Omron Sysmac Studio project comodo-sync-lib (Sysmac Studio 1.64.0.64008, LibraryProject)

# Controller new_Controller_0: NX102-9020 version 1.50
Task PrimaryTask (priority 4, period or condition 2000): Program0

VAR_GLOBAL
    Robot_Positions : ARRAY[0..5] OF LREAL;
    Robot_In : LWORD;  (* network input *)
    Robot_Out : LWORD;  (* network output *)
    In_Joint_1 : LREAL;  (* published *)
    In_Joint_2 : LREAL;  (* published *)
    In_Joint_3 : LREAL;  (* published *)
    In_Joint_4 : LREAL;  (* published *)
    In_Joint_5 : LREAL;  (* published *)
    In_Joint_6 : LREAL;  (* published *)
    Out_Joint_1 : LREAL;  (* published *)
    Out_Joint_2 : LREAL;  (* published *)
    Out_Joint_3 : LREAL;  (* published *)
    Out_Joint_4 : LREAL;  (* published *)
    Out_Joint_5 : LREAL;  (* published *)
    Out_Joint_6 : LREAL;  (* published *)
    Is_Monitoring : BOOL;
    Is_Moving_Linear : BOOL;
END_VAR

PROGRAM Program0
VAR
    test : BOOL;
END_VAR

(* Section Section0: ladder, written here as Structured Text *)

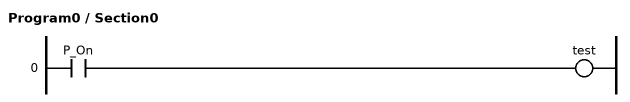
(* Rung 0 *)
test := P_On;
END_PROGRAM

FUNCTION MapLREAL : LREAL
VAR_INPUT
    Num : LREAL;
    In_Min : LREAL;
    In_Max : LREAL;
    Out_Min : LREAL;
    Out_Max : LREAL;
END_VAR
MapLREAL := (Num - In_Min) * (Out_Max - Out_Min) / (In_Max - In_Min) + Out_Min;
END_FUNCTION

FUNCTION ReceiveRobotPositions : BOOL
VAR_EXTERNAL
    Robot_Positions : ARRAY[0..5] OF LREAL;
    In_Joint_1 : LREAL;
    In_Joint_2 : LREAL;
    In_Joint_3 : LREAL;
    In_Joint_4 : LREAL;
    In_Joint_5 : LREAL;
    In_Joint_6 : LREAL;
END_VAR
IF In_Joint_1 <> Robot_Positions[0] THEN
	In_Joint_1 := Robot_Positions[0];
END_IF;
IF In_Joint_2 <> Robot_Positions[1] THEN
	In_Joint_2 := Robot_Positions[1];
END_IF;
IF In_Joint_3 <> Robot_Positions[2] THEN
	In_Joint_3 := Robot_Positions[2];
END_IF;
IF In_Joint_4 <> Robot_Positions[3] THEN
	In_Joint_4 := Robot_Positions[3];
END_IF;
IF In_Joint_5 <> Robot_Positions[4] THEN
	In_Joint_5 := Robot_Positions[4];
END_IF;
IF In_Joint_6 <> Robot_Positions[5] THEN
	In_Joint_6 := Robot_Positions[5];
END_IF;
END_FUNCTION

FUNCTION SendPositionsToRobot : BOOL
VAR
    Temp_Output : LWORD;
    Temp_Bits : LWORD;
    Shifted_Bits : LWORD;
END_VAR
VAR CONSTANT
    Movement_Bit : LWORD := 16#2000000000000000;
    Monitor_Bit : LWORD := 16#1000000000000000;
END_VAR
VAR_EXTERNAL
    Robot_Positions : ARRAY[0..5] OF LREAL;
    Robot_In : LWORD;
    Out_Joint_1 : LREAL;
    Out_Joint_2 : LREAL;
    Out_Joint_3 : LREAL;
    Out_Joint_4 : LREAL;
    Out_Joint_5 : LREAL;
    Out_Joint_6 : LREAL;
    Is_Moving_Linear : BOOL;
    Is_Monitoring : BOOL;
END_VAR
Robot_Positions[0] := Out_Joint_1;
Robot_Positions[1] := Out_Joint_2;
Robot_Positions[2] := Out_Joint_3;
Robot_Positions[3] := Out_Joint_4;
Robot_Positions[4] := Out_Joint_5;
Robot_Positions[5] := Out_Joint_6;

Temp_Output := 16#0;

Temp_Bits := LREAL_TO_LWORD(MapLREAL(Robot_Positions[0], -230.0, 230.0, 0.0, 1023.0));
Temp_Output := Temp_Output OR Temp_Bits;


Temp_Bits := LREAL_TO_LWORD(MapLREAL(Robot_Positions[1], -115.0, 113.0, 0.0, 1023.0));
Shifted_Bits := SHL(Temp_Bits, 10);
Temp_Output := Temp_Output OR Shifted_Bits;


Temp_Bits := LREAL_TO_LWORD(MapLREAL(Robot_Positions[2], -205.0, 55.0, 0.0, 1023.0));
Shifted_Bits := SHL(Temp_Bits, 20);
Temp_Output := Temp_Output OR Shifted_Bits;


Temp_Bits := LREAL_TO_LWORD(MapLREAL(Robot_Positions[3], -230.0, 230.0, 0.0, 1023.0));
Shifted_Bits := SHL(Temp_Bits, 30);
Temp_Output := Temp_Output OR Shifted_Bits;


Temp_Bits := LREAL_TO_LWORD(MapLREAL(Robot_Positions[4], -125.0, 120.0, 0.0, 1023.0));
Shifted_Bits := SHL(Temp_Bits, 40);
Temp_Output := Temp_Output OR Shifted_Bits;


Temp_Bits := LREAL_TO_LWORD(MapLREAL(Robot_Positions[5], -400.0, 400.0, 0.0, 1023.0));
Shifted_Bits := SHL(Temp_Bits, 50);
Temp_Output := Temp_Output OR Shifted_Bits;

IF Is_Monitoring THEN 
		Temp_Output := Temp_Output OR Monitor_Bit;
ELSE
		Temp_Output := Temp_Output AND (NOT Monitor_Bit);
END_IF;

IF Is_Moving_Linear THEN
		Temp_Output := Temp_Output OR Movement_Bit;
ELSE
		Temp_Output := Temp_Output AND (NOT Movement_Bit);
END_IF;

Robot_In := Temp_Output;
END_FUNCTION

FUNCTION ChangeState : BOOL
VAR
    Previous_Monitor_State : BOOL;
    Temp_Output : LWORD;
END_VAR
VAR CONSTANT
    Monitor_Bit : LWORD := 16#1000000000000000;
END_VAR
VAR
    Previous_Movement_State : BOOL;
END_VAR
VAR CONSTANT
    Movement_Bit : LWORD := 16#2000000000000000;
END_VAR
VAR_EXTERNAL
    Is_Monitoring : BOOL;
    Robot_Out : LWORD;
    Robot_In : LWORD;
    Is_Moving_Linear : BOOL;
END_VAR
IF Is_Monitoring <> Previous_Monitor_State OR Is_Moving_Linear <> Previous_Movement_State THEN
	Temp_Output := Robot_In;
	IF Is_Monitoring THEN 
		Temp_Output := Temp_Output OR Monitor_Bit;
	ELSE
		Temp_Output := Temp_Output AND (NOT Monitor_Bit);
	END_IF;
	
	IF Is_Moving_Linear THEN
		Temp_Output := Temp_Output OR Movement_Bit;
	ELSE
		Temp_Output := Temp_Output AND (NOT Movement_Bit);
	END_IF;
		
	Previous_Monitor_State := Is_Monitoring;
	Previous_Movement_State := Is_Moving_Linear;
	
	Robot_In := Temp_Output;
END_IF;
END_FUNCTION

FUNCTION_BLOCK ParseRobotData
VAR
    value : UINT;
    shifted_input : LWORD;
END_VAR
VAR_INPUT
    IN : BOOL;
END_VAR
VAR_EXTERNAL
    Robot_Positions : ARRAY[0..5] OF LREAL;
    Robot_Out : LWORD;
END_VAR
value := LWORD_TO_UINT(Robot_Out AND LWORD#16#3FF);
Robot_Positions[0] :=MapLREAL(value, 0.0, 1023.0, -230.0, 230.0);

shifted_input := SHR(Robot_Out, 10);
value := LWORD_TO_UINT(shifted_input AND LWORD#16#3FF);
Robot_Positions[1]:=MapLREAL(value, 0.0, 1023.0, -115.0, 113.0);

shifted_input := SHR(Robot_Out, 20);
value := LWORD_TO_UINT(shifted_input AND LWORD#16#3FF);
Robot_Positions[2]:=MapLREAL(value, 0.0, 1023.0, -205.0, 55.0);

shifted_input := SHR(Robot_Out, 30);
value := LWORD_TO_UINT(shifted_input AND LWORD#16#3FF);
Robot_Positions[3]:=MapLREAL(value, 0.0, 1023.0, -230.0, 230.0);

shifted_input := SHR(Robot_Out, 40);
value := LWORD_TO_UINT(shifted_input AND LWORD#16#3FF);
Robot_Positions[4]:=MapLREAL(value, 0.0, 1023.0, -125.0, 120.0);

shifted_input := SHR(Robot_Out, 50);
value := LWORD_TO_UINT(shifted_input AND LWORD#16#3FF);
Robot_Positions[5]:=MapLREAL(value, 0.0, 1023.0, -400.0, 400.0);
END_FUNCTION_BLOCK